  gc_ErrTranslation_fr_Texts : ARRAY[0..1193] OF POINTER TO WSTRING(101) := [ADR(gc_ErrTranslation_fr_Text0), ADR(gc_ErrTranslation_fr_Text1), ADR(gc_ErrTranslation_fr_Text2), ADR(gc_ErrTranslation_fr_Text3), ADR(gc_ErrTranslation_fr_Text4), ADR(gc_ErrTranslation_fr_Text5), ADR(gc_ErrTranslation_fr_Text6), ADR(gc_ErrTranslation_fr_Text7), ADR(gc_ErrTranslation_fr_Text8), ADR(gc_ErrTranslation_fr_Text9), ADR(gc_ErrTranslation_fr_Text10), ADR(gc_ErrTranslation_fr_Text11), ADR(gc_ErrTranslation_fr_Text12), ADR(gc_ErrTranslation_fr_Text13), ADR(gc_ErrTranslation_fr_Text14), ADR(gc_ErrTranslation_fr_Text15), ADR(gc_ErrTranslation_fr_Text16), ADR(gc_ErrTranslation_fr_Text17), ADR(gc_ErrTranslation_fr_Text18), ADR(gc_ErrTranslation_fr_Text19), ADR(gc_ErrTranslation_fr_Text20), ADR(gc_ErrTranslation_fr_Text21), ADR(gc_ErrTranslation_fr_Text22), ADR(gc_ErrTranslation_fr_Text23), ADR(gc_ErrTranslation_fr_Text24), ADR(gc_ErrTranslation_fr_Text25), ADR(gc_ErrTranslation_fr_Text26), ADR(gc_ErrTranslation_fr_Text27), ADR(gc_ErrTranslation_fr_Text28), ADR(gc_ErrTranslation_fr_Text29), ADR(gc_ErrTranslation_fr_Text30), ADR(gc_ErrTranslation_fr_Text31), ADR(gc_ErrTranslation_fr_Text32), ADR(gc_ErrTranslation_fr_Text33), ADR(gc_ErrTranslation_fr_Text34), ADR(gc_ErrTranslation_fr_Text35), ADR(gc_ErrTranslation_fr_Text36), ADR(gc_ErrTranslation_fr_Text37), ADR(gc_ErrTranslation_fr_Text38), ADR(gc_ErrTranslation_fr_Text39), ADR(gc_ErrTranslation_fr_Text40), ADR(gc_ErrTranslation_fr_Text41), ADR(gc_ErrTranslation_fr_Text42), ADR(gc_ErrTranslation_fr_Text43), ADR(gc_ErrTranslation_fr_Text44), ADR(gc_ErrTranslation_fr_Text45), ADR(gc_ErrTranslation_fr_Text46), ADR(gc_ErrTranslation_fr_Text47), ADR(gc_ErrTranslation_fr_Text48), ADR(gc_ErrTranslation_fr_Text49), ADR(gc_ErrTranslation_fr_Text50), ADR(gc_ErrTranslation_fr_Text51), ADR(gc_ErrTranslation_fr_Text52), ADR(gc_ErrTranslation_fr_Text53), ADR(gc_ErrTranslation_fr_Text54), ADR(gc_ErrTranslation_fr_Text55), ADR(gc_ErrTranslation_fr_Text56), ADR(gc_ErrTranslation_fr_Text57), ADR(gc_ErrTranslation_fr_Text58), ADR(gc_ErrTranslation_fr_Text59), ADR(gc_ErrTranslation_fr_Text60), ADR(gc_ErrTranslation_fr_Text61), ADR(gc_ErrTranslation_fr_Text62), ADR(gc_ErrTranslation_fr_Text63), ADR(gc_ErrTranslation_fr_Text64), ADR(gc_ErrTranslation_fr_Text65), ADR(gc_ErrTranslation_fr_Text66), ADR(gc_ErrTranslation_fr_Text67), ADR(gc_ErrTranslation_fr_Text68), ADR(gc_ErrTranslation_fr_Text69), ADR(gc_ErrTranslation_fr_Text70), ADR(gc_ErrTranslation_fr_Text71), ADR(gc_ErrTranslation_fr_Text72), ADR(gc_ErrTranslation_fr_Text73), ADR(gc_ErrTranslation_fr_Text74), ADR(gc_ErrTranslation_fr_Text75), ADR(gc_ErrTranslation_fr_Text76), ADR(gc_ErrTranslation_fr_Text77), ADR(gc_ErrTranslation_fr_Text78), ADR(gc_ErrTranslation_fr_Text79), ADR(gc_ErrTranslation_fr_Text80), ADR(gc_ErrTranslation_fr_Text81), ADR(gc_ErrTranslation_fr_Text82), ADR(gc_ErrTranslation_fr_Text83), ADR(gc_ErrTranslation_fr_Text84), ADR(gc_ErrTranslation_fr_Text85), ADR(gc_ErrTranslation_fr_Text86), ADR(gc_ErrTranslation_fr_Text87), ADR(gc_ErrTranslation_fr_Text88), ADR(gc_ErrTranslation_fr_Text89), ADR(gc_ErrTranslation_fr_Text90), ADR(gc_ErrTranslation_fr_Text91), ADR(gc_ErrTranslation_fr_Text92), ADR(gc_ErrTranslation_fr_Text93), ADR(gc_ErrTranslation_fr_Text94), ADR(gc_ErrTranslation_fr_Text95), ADR(gc_ErrTranslation_fr_Text96), ADR(gc_ErrTranslation_fr_Text97), ADR(gc_ErrTranslation_fr_Text98), ADR(gc_ErrTranslation_fr_Text99), ADR(gc_ErrTranslation_fr_Text100), ADR(gc_ErrTranslation_fr_Text101), ADR(gc_ErrTranslation_fr_Text102), ADR(gc_ErrTranslation_fr_Text103), ADR(gc_ErrTranslation_fr_Text104), ADR(gc_ErrTranslation_fr_Text105), ADR(gc_ErrTranslation_fr_Text106), ADR(gc_ErrTranslation_fr_Text107), ADR(gc_ErrTranslation_fr_Text108), ADR(gc_ErrTranslation_fr_Text109), ADR(gc_ErrTranslation_fr_Text110), ADR(gc_ErrTranslation_fr_Text111), ADR(gc_ErrTranslation_fr_Text112), ADR(gc_ErrTranslation_fr_Text113), ADR(gc_ErrTranslation_fr_Text114), ADR(gc_ErrTranslation_fr_Text115), ADR(gc_ErrTranslation_fr_Text116), ADR(gc_ErrTranslation_fr_Text117), ADR(gc_ErrTranslation_fr_Text118), ADR(gc_ErrTranslation_fr_Text119), ADR(gc_ErrTranslation_fr_Text120), ADR(gc_ErrTranslation_fr_Text121), ADR(gc_ErrTranslation_fr_Text122), ADR(gc_ErrTranslation_fr_Text123), ADR(gc_ErrTranslation_fr_Text124), ADR(gc_ErrTranslation_fr_Text125), ADR(gc_ErrTranslation_fr_Text126), ADR(gc_ErrTranslation_fr_Text127), ADR(gc_ErrTranslation_fr_Text128), ADR(gc_ErrTranslation_fr_Text129), ADR(gc_ErrTranslation_fr_Text130), ADR(gc_ErrTranslation_fr_Text131), ADR(gc_ErrTranslation_fr_Text132), ADR(gc_ErrTranslation_fr_Text133), ADR(gc_ErrTranslation_fr_Text134), ADR(gc_ErrTranslation_fr_Text135), ADR(gc_ErrTranslation_fr_Text136), ADR(gc_ErrTranslation_fr_Text137), ADR(gc_ErrTranslation_fr_Text138), ADR(gc_ErrTranslation_fr_Text139), ADR(gc_ErrTranslation_fr_Text140), ADR(gc_ErrTranslation_fr_Text141), ADR(gc_ErrTranslation_fr_Text142), ADR(gc_ErrTranslation_fr_Text143), ADR(gc_ErrTranslation_fr_Text144), ADR(gc_ErrTranslation_fr_Text145), ADR(gc_ErrTranslation_fr_Text146), ADR(gc_ErrTranslation_fr_Text147), ADR(gc_ErrTranslation_fr_Text148), ADR(gc_ErrTranslation_fr_Text149), ADR(gc_ErrTranslation_fr_Text150), ADR(gc_ErrTranslation_fr_Text151), ADR(gc_ErrTranslation_fr_Text152), ADR(gc_ErrTranslation_fr_Text153), ADR(gc_ErrTranslation_fr_Text154), ADR(gc_ErrTranslation_fr_Text155), ADR(gc_ErrTranslation_fr_Text156), ADR(gc_ErrTranslation_fr_Text157), ADR(gc_ErrTranslation_fr_Text158), ADR(gc_ErrTranslation_fr_Text159), ADR(gc_ErrTranslation_fr_Text160), ADR(gc_ErrTranslation_fr_Text161), ADR(gc_ErrTranslation_fr_Text162), ADR(gc_ErrTranslation_fr_Text163), ADR(gc_ErrTranslation_fr_Text164), ADR(gc_ErrTranslation_fr_Text165), ADR(gc_ErrTranslation_fr_Text166), ADR(gc_ErrTranslation_fr_Text167), ADR(gc_ErrTranslation_fr_Text168), ADR(gc_ErrTranslation_fr_Text169), ADR(gc_ErrTranslation_fr_Text170), ADR(gc_ErrTranslation_fr_Text171), ADR(gc_ErrTranslation_fr_Text172), ADR(gc_ErrTranslation_fr_Text173), ADR(gc_ErrTranslation_fr_Text174), ADR(gc_ErrTranslation_fr_Text175), ADR(gc_ErrTranslation_fr_Text176), ADR(gc_ErrTranslation_fr_Text177), ADR(gc_ErrTranslation_fr_Text178), ADR(gc_ErrTranslation_fr_Text179), ADR(gc_ErrTranslation_fr_Text180), ADR(gc_ErrTranslation_fr_Text181), ADR(gc_ErrTranslation_fr_Text182), ADR(gc_ErrTranslation_fr_Text183), ADR(gc_ErrTranslation_fr_Text184), ADR(gc_ErrTranslation_fr_Text185), ADR(gc_ErrTranslation_fr_Text186), ADR(gc_ErrTranslation_fr_Text187), ADR(gc_ErrTranslation_fr_Text188), ADR(gc_ErrTranslation_fr_Text189), ADR(gc_ErrTranslation_fr_Text190), ADR(gc_ErrTranslation_fr_Text191), ADR(gc_ErrTranslation_fr_Text192), ADR(gc_ErrTranslation_fr_Text193), ADR(gc_ErrTranslation_fr_Text194), ADR(gc_ErrTranslation_fr_Text195), ADR(gc_ErrTranslation_fr_Text196), ADR(gc_ErrTranslation_fr_Text197), ADR(gc_ErrTranslation_fr_Text198), ADR(gc_ErrTranslation_fr_Text199), ADR(gc_ErrTranslation_fr_Text200), ADR(gc_ErrTranslation_fr_Text201), ADR(gc_ErrTranslation_fr_Text202), ADR(gc_ErrTranslation_fr_Text203), ADR(gc_ErrTranslation_fr_Text204), ADR(gc_ErrTranslation_fr_Text205), ADR(gc_ErrTranslation_fr_Text206), ADR(gc_ErrTranslation_fr_Text207), ADR(gc_ErrTranslation_fr_Text208), ADR(gc_ErrTranslation_fr_Text209), ADR(gc_ErrTranslation_fr_Text210), ADR(gc_ErrTranslation_fr_Text211), ADR(gc_ErrTranslation_fr_Text212), ADR(gc_ErrTranslation_fr_Text213), ADR(gc_ErrTranslation_fr_Text214), ADR(gc_ErrTranslation_fr_Text215), ADR(gc_ErrTranslation_fr_Text216), ADR(gc_ErrTranslation_fr_Text217), ADR(gc_ErrTranslation_fr_Text218), ADR(gc_ErrTranslation_fr_Text219), ADR(gc_ErrTranslation_fr_Text220), ADR(gc_ErrTranslation_fr_Text221), ADR(gc_ErrTranslation_fr_Text222), ADR(gc_ErrTranslation_fr_Text223), ADR(gc_ErrTranslation_fr_Text224), ADR(gc_ErrTranslation_fr_Text225), ADR(gc_ErrTranslation_fr_Text226), ADR(gc_ErrTranslation_fr_Text227), ADR(gc_ErrTranslation_fr_Text228), ADR(gc_ErrTranslation_fr_Text229), ADR(gc_ErrTranslation_fr_Text230), ADR(gc_ErrTranslation_fr_Text231), ADR(gc_ErrTranslation_fr_Text232), ADR(gc_ErrTranslation_fr_Text233), ADR(gc_ErrTranslation_fr_Text234), ADR(gc_ErrTranslation_fr_Text235), ADR(gc_ErrTranslation_fr_Text236), ADR(gc_ErrTranslation_fr_Text237), ADR(gc_ErrTranslation_fr_Text238), ADR(gc_ErrTranslation_fr_Text239), ADR(gc_ErrTranslation_fr_Text240), ADR(gc_ErrTranslation_fr_Text241), ADR(gc_ErrTranslation_fr_Text242), ADR(gc_ErrTranslation_fr_Text243), ADR(gc_ErrTranslation_fr_Text244), ADR(gc_ErrTranslation_fr_Text245), ADR(gc_ErrTranslation_fr_Text246), ADR(gc_ErrTranslation_fr_Text247), ADR(gc_ErrTranslation_fr_Text248), ADR(gc_ErrTranslation_fr_Text249), ADR(gc_ErrTranslation_fr_Text250), ADR(gc_ErrTranslation_fr_Text251), ADR(gc_ErrTranslation_fr_Text252), ADR(gc_ErrTranslation_fr_Text253), ADR(gc_ErrTranslation_fr_Text254), ADR(gc_ErrTranslation_fr_Text255), ADR(gc_ErrTranslation_fr_Text256), ADR(gc_ErrTranslation_fr_Text257), ADR(gc_ErrTranslation_fr_Text258), ADR(gc_ErrTranslation_fr_Text259), ADR(gc_ErrTranslation_fr_Text260), ADR(gc_ErrTranslation_fr_Text261), ADR(gc_ErrTranslation_fr_Text262), ADR(gc_ErrTranslation_fr_Text263), ADR(gc_ErrTranslation_fr_Text264), ADR(gc_ErrTranslation_fr_Text265), ADR(gc_ErrTranslation_fr_Text266), ADR(gc_ErrTranslation_fr_Text267), ADR(gc_ErrTranslation_fr_Text268), ADR(gc_ErrTranslation_fr_Text269), ADR(gc_ErrTranslation_fr_Text270), ADR(gc_ErrTranslation_fr_Text271), ADR(gc_ErrTranslation_fr_Text272), ADR(gc_ErrTranslation_fr_Text273), ADR(gc_ErrTranslation_fr_Text274), ADR(gc_ErrTranslation_fr_Text275), ADR(gc_ErrTranslation_fr_Text276), ADR(gc_ErrTranslation_fr_Text277), ADR(gc_ErrTranslation_fr_Text278), ADR(gc_ErrTranslation_fr_Text279), ADR(gc_ErrTranslation_fr_Text280), ADR(gc_ErrTranslation_fr_Text281), ADR(gc_ErrTranslation_fr_Text282), ADR(gc_ErrTranslation_fr_Text283), ADR(gc_ErrTranslation_fr_Text284), ADR(gc_ErrTranslation_fr_Text285), ADR(gc_ErrTranslation_fr_Text286), ADR(gc_ErrTranslation_fr_Text287), ADR(gc_ErrTranslation_fr_Text288), ADR(gc_ErrTranslation_fr_Text289), ADR(gc_ErrTranslation_fr_Text290), ADR(gc_ErrTranslation_fr_Text291), ADR(gc_ErrTranslation_fr_Text292), ADR(gc_ErrTranslation_fr_Text293), ADR(gc_ErrTranslation_fr_Text294), ADR(gc_ErrTranslation_fr_Text295), ADR(gc_ErrTranslation_fr_Text296), ADR(gc_ErrTranslation_fr_Text297), ADR(gc_ErrTranslation_fr_Text298), ADR(gc_ErrTranslation_fr_Text299), ADR(gc_ErrTranslation_fr_Text300), ADR(gc_ErrTranslation_fr_Text301), ADR(gc_ErrTranslation_fr_Text302), ADR(gc_ErrTranslation_fr_Text303), ADR(gc_ErrTranslation_fr_Text304), ADR(gc_ErrTranslation_fr_Text305), ADR(gc_ErrTranslation_fr_Text306), ADR(gc_ErrTranslation_fr_Text307), ADR(gc_ErrTranslation_fr_Text308), ADR(gc_ErrTranslation_fr_Text309), ADR(gc_ErrTranslation_fr_Text310), ADR(gc_ErrTranslation_fr_Text311), ADR(gc_ErrTranslation_fr_Text312), ADR(gc_ErrTranslation_fr_Text313), ADR(gc_ErrTranslation_fr_Text314), ADR(gc_ErrTranslation_fr_Text315), ADR(gc_ErrTranslation_fr_Text316), ADR(gc_ErrTranslation_fr_Text317), ADR(gc_ErrTranslation_fr_Text318), ADR(gc_ErrTranslation_fr_Text319), ADR(gc_ErrTranslation_fr_Text320), ADR(gc_ErrTranslation_fr_Text321), ADR(gc_ErrTranslation_fr_Text322), ADR(gc_ErrTranslation_fr_Text323), ADR(gc_ErrTranslation_fr_Text324), ADR(gc_ErrTranslation_fr_Text325), ADR(gc_ErrTranslation_fr_Text326), ADR(gc_ErrTranslation_fr_Text327), ADR(gc_ErrTranslation_fr_Text328), ADR(gc_ErrTranslation_fr_Text329), ADR(gc_ErrTranslation_fr_Text330), ADR(gc_ErrTranslation_fr_Text331), ADR(gc_ErrTranslation_fr_Text332), ADR(gc_ErrTranslation_fr_Text333), ADR(gc_ErrTranslation_fr_Text334), ADR(gc_ErrTranslation_fr_Text335), ADR(gc_ErrTranslation_fr_Text336), ADR(gc_ErrTranslation_fr_Text337), ADR(gc_ErrTranslation_fr_Text338), ADR(gc_ErrTranslation_fr_Text339), ADR(gc_ErrTranslation_fr_Text340), ADR(gc_ErrTranslation_fr_Text341), ADR(gc_ErrTranslation_fr_Text342), ADR(gc_ErrTranslation_fr_Text343), ADR(gc_ErrTranslation_fr_Text344), ADR(gc_ErrTranslation_fr_Text345), ADR(gc_ErrTranslation_fr_Text346), ADR(gc_ErrTranslation_fr_Text347), ADR(gc_ErrTranslation_fr_Text348), ADR(gc_ErrTranslation_fr_Text349), ADR(gc_ErrTranslation_fr_Text350), ADR(gc_ErrTranslation_fr_Text351), ADR(gc_ErrTranslation_fr_Text352), ADR(gc_ErrTranslation_fr_Text353), ADR(gc_ErrTranslation_fr_Text354), ADR(gc_ErrTranslation_fr_Text355), ADR(gc_ErrTranslation_fr_Text356), ADR(gc_ErrTranslation_fr_Text357), ADR(gc_ErrTranslation_fr_Text358), ADR(gc_ErrTranslation_fr_Text359), ADR(gc_ErrTranslation_fr_Text360), ADR(gc_ErrTranslation_fr_Text361), ADR(gc_ErrTranslation_fr_Text362), ADR(gc_ErrTranslation_fr_Text363), ADR(gc_ErrTranslation_fr_Text364), ADR(gc_ErrTranslation_fr_Text365), ADR(gc_ErrTranslation_fr_Text366), ADR(gc_ErrTranslation_fr_Text367), ADR(gc_ErrTranslation_fr_Text368), ADR(gc_ErrTranslation_fr_Text369), ADR(gc_ErrTranslation_fr_Text370), ADR(gc_ErrTranslation_fr_Text371), ADR(gc_ErrTranslation_fr_Text372), ADR(gc_ErrTranslation_fr_Text373), ADR(gc_ErrTranslation_fr_Text374), ADR(gc_ErrTranslation_fr_Text375), ADR(gc_ErrTranslation_fr_Text376), ADR(gc_ErrTranslation_fr_Text377), ADR(gc_ErrTranslation_fr_Text378), ADR(gc_ErrTranslation_fr_Text379), ADR(gc_ErrTranslation_fr_Text380), ADR(gc_ErrTranslation_fr_Text381), ADR(gc_ErrTranslation_fr_Text382), ADR(gc_ErrTranslation_fr_Text383), ADR(gc_ErrTranslation_fr_Text384), ADR(gc_ErrTranslation_fr_Text385), ADR(gc_ErrTranslation_fr_Text386), ADR(gc_ErrTranslation_fr_Text387), ADR(gc_ErrTranslation_fr_Text388), ADR(gc_ErrTranslation_fr_Text389), ADR(gc_ErrTranslation_fr_Text390), ADR(gc_ErrTranslation_fr_Text391), ADR(gc_ErrTranslation_fr_Text392), ADR(gc_ErrTranslation_fr_Text393), ADR(gc_ErrTranslation_fr_Text394), ADR(gc_ErrTranslation_fr_Text395), ADR(gc_ErrTranslation_fr_Text396), ADR(gc_ErrTranslation_fr_Text397), ADR(gc_ErrTranslation_fr_Text398), ADR(gc_ErrTranslation_fr_Text399), ADR(gc_ErrTranslation_fr_Text400), ADR(gc_ErrTranslation_fr_Text401), ADR(gc_ErrTranslation_fr_Text402), ADR(gc_ErrTranslation_fr_Text403), ADR(gc_ErrTranslation_fr_Text404), ADR(gc_ErrTranslation_fr_Text405), ADR(gc_ErrTranslation_fr_Text406), ADR(gc_ErrTranslation_fr_Text407), ADR(gc_ErrTranslation_fr_Text408), ADR(gc_ErrTranslation_fr_Text409), ADR(gc_ErrTranslation_fr_Text410), ADR(gc_ErrTranslation_fr_Text411), ADR(gc_ErrTranslation_fr_Text412), ADR(gc_ErrTranslation_fr_Text413), ADR(gc_ErrTranslation_fr_Text414), ADR(gc_ErrTranslation_fr_Text415), ADR(gc_ErrTranslation_fr_Text416), ADR(gc_ErrTranslation_fr_Text417), ADR(gc_ErrTranslation_fr_Text418), ADR(gc_ErrTranslation_fr_Text419), ADR(gc_ErrTranslation_fr_Text420), ADR(gc_ErrTranslation_fr_Text421), ADR(gc_ErrTranslation_fr_Text422), ADR(gc_ErrTranslation_fr_Text423), ADR(gc_ErrTranslation_fr_Text424), ADR(gc_ErrTranslation_fr_Text425), ADR(gc_ErrTranslation_fr_Text426), ADR(gc_ErrTranslation_fr_Text427), ADR(gc_ErrTranslation_fr_Text428), ADR(gc_ErrTranslation_fr_Text429), ADR(gc_ErrTranslation_fr_Text430), ADR(gc_ErrTranslation_fr_Text431), ADR(gc_ErrTranslation_fr_Text432), ADR(gc_ErrTranslation_fr_Text433), ADR(gc_ErrTranslation_fr_Text434), ADR(gc_ErrTranslation_fr_Text435), ADR(gc_ErrTranslation_fr_Text436), ADR(gc_ErrTranslation_fr_Text437), ADR(gc_ErrTranslation_fr_Text438), ADR(gc_ErrTranslation_fr_Text439), ADR(gc_ErrTranslation_fr_Text440), ADR(gc_ErrTranslation_fr_Text441), ADR(gc_ErrTranslation_fr_Text442), ADR(gc_ErrTranslation_fr_Text443), ADR(gc_ErrTranslation_fr_Text444), ADR(gc_ErrTranslation_fr_Text445), ADR(gc_ErrTranslation_fr_Text446), ADR(gc_ErrTranslation_fr_Text447), ADR(gc_ErrTranslation_fr_Text448), ADR(gc_ErrTranslation_fr_Text449), ADR(gc_ErrTranslation_fr_Text450), ADR(gc_ErrTranslation_fr_Text451), ADR(gc_ErrTranslation_fr_Text452), ADR(gc_ErrTranslation_fr_Text453), ADR(gc_ErrTranslation_fr_Text454), ADR(gc_ErrTranslation_fr_Text455), ADR(gc_ErrTranslation_fr_Text456), ADR(gc_ErrTranslation_fr_Text457), ADR(gc_ErrTranslation_fr_Text458), ADR(gc_ErrTranslation_fr_Text459), ADR(gc_ErrTranslation_fr_Text460), ADR(gc_ErrTranslation_fr_Text461), ADR(gc_ErrTranslation_fr_Text462), ADR(gc_ErrTranslation_fr_Text463), ADR(gc_ErrTranslation_fr_Text464), ADR(gc_ErrTranslation_fr_Text465), ADR(gc_ErrTranslation_fr_Text466), ADR(gc_ErrTranslation_fr_Text467), ADR(gc_ErrTranslation_fr_Text468), ADR(gc_ErrTranslation_fr_Text469), ADR(gc_ErrTranslation_fr_Text470), ADR(gc_ErrTranslation_fr_Text471), ADR(gc_ErrTranslation_fr_Text472), ADR(gc_ErrTranslation_fr_Text473), ADR(gc_ErrTranslation_fr_Text474), ADR(gc_ErrTranslation_fr_Text475), ADR(gc_ErrTranslation_fr_Text476), ADR(gc_ErrTranslation_fr_Text477), ADR(gc_ErrTranslation_fr_Text478), ADR(gc_ErrTranslation_fr_Text479), ADR(gc_ErrTranslation_fr_Text480), ADR(gc_ErrTranslation_fr_Text481), ADR(gc_ErrTranslation_fr_Text482), ADR(gc_ErrTranslation_fr_Text483), ADR(gc_ErrTranslation_fr_Text484), ADR(gc_ErrTranslation_fr_Text485), ADR(gc_ErrTranslation_fr_Text486), ADR(gc_ErrTranslation_fr_Text487), ADR(gc_ErrTranslation_fr_Text488), ADR(gc_ErrTranslation_fr_Text489), ADR(gc_ErrTranslation_fr_Text490), ADR(gc_ErrTranslation_fr_Text491), ADR(gc_ErrTranslation_fr_Text492), ADR(gc_ErrTranslation_fr_Text493), ADR(gc_ErrTranslation_fr_Text494), ADR(gc_ErrTranslation_fr_Text495), ADR(gc_ErrTranslation_fr_Text496), ADR(gc_ErrTranslation_fr_Text497), ADR(gc_ErrTranslation_fr_Text498), ADR(gc_ErrTranslation_fr_Text499), ADR(gc_ErrTranslation_fr_Text500), ADR(gc_ErrTranslation_fr_Text501), ADR(gc_ErrTranslation_fr_Text502), ADR(gc_ErrTranslation_fr_Text503), ADR(gc_ErrTranslation_fr_Text504), ADR(gc_ErrTranslation_fr_Text505), ADR(gc_ErrTranslation_fr_Text506), ADR(gc_ErrTranslation_fr_Text507), ADR(gc_ErrTranslation_fr_Text508), ADR(gc_ErrTranslation_fr_Text509), ADR(gc_ErrTranslation_fr_Text510), ADR(gc_ErrTranslation_fr_Text511), ADR(gc_ErrTranslation_fr_Text512), ADR(gc_ErrTranslation_fr_Text513), ADR(gc_ErrTranslation_fr_Text514), ADR(gc_ErrTranslation_fr_Text515), ADR(gc_ErrTranslation_fr_Text516), ADR(gc_ErrTranslation_fr_Text517), ADR(gc_ErrTranslation_fr_Text518), ADR(gc_ErrTranslation_fr_Text519), ADR(gc_ErrTranslation_fr_Text520), ADR(gc_ErrTranslation_fr_Text521), ADR(gc_ErrTranslation_fr_Text522), ADR(gc_ErrTranslation_fr_Text523), ADR(gc_ErrTranslation_fr_Text524), ADR(gc_ErrTranslation_fr_Text525), ADR(gc_ErrTranslation_fr_Text526), ADR(gc_ErrTranslation_fr_Text527), ADR(gc_ErrTranslation_fr_Text528), ADR(gc_ErrTranslation_fr_Text529), ADR(gc_ErrTranslation_fr_Text530), ADR(gc_ErrTranslation_fr_Text531), ADR(gc_ErrTranslation_fr_Text532), ADR(gc_ErrTranslation_fr_Text533), ADR(gc_ErrTranslation_fr_Text534), ADR(gc_ErrTranslation_fr_Text535), ADR(gc_ErrTranslation_fr_Text536), ADR(gc_ErrTranslation_fr_Text537), ADR(gc_ErrTranslation_fr_Text538), ADR(gc_ErrTranslation_fr_Text539), ADR(gc_ErrTranslation_fr_Text540), ADR(gc_ErrTranslation_fr_Text541), ADR(gc_ErrTranslation_fr_Text542), ADR(gc_ErrTranslation_fr_Text543), ADR(gc_ErrTranslation_fr_Text544), ADR(gc_ErrTranslation_fr_Text545), ADR(gc_ErrTranslation_fr_Text546), ADR(gc_ErrTranslation_fr_Text547), ADR(gc_ErrTranslation_fr_Text548), ADR(gc_ErrTranslation_fr_Text549), ADR(gc_ErrTranslation_fr_Text550), ADR(gc_ErrTranslation_fr_Text551), ADR(gc_ErrTranslation_fr_Text552), ADR(gc_ErrTranslation_fr_Text553), ADR(gc_ErrTranslation_fr_Text554), ADR(gc_ErrTranslation_fr_Text555), ADR(gc_ErrTranslation_fr_Text556), ADR(gc_ErrTranslation_fr_Text557), ADR(gc_ErrTranslation_fr_Text558), ADR(gc_ErrTranslation_fr_Text559), ADR(gc_ErrTranslation_fr_Text560), ADR(gc_ErrTranslation_fr_Text561), ADR(gc_ErrTranslation_fr_Text562), ADR(gc_ErrTranslation_fr_Text563), ADR(gc_ErrTranslation_fr_Text564), ADR(gc_ErrTranslation_fr_Text565), ADR(gc_ErrTranslation_fr_Text566), ADR(gc_ErrTranslation_fr_Text567), ADR(gc_ErrTranslation_fr_Text568), ADR(gc_ErrTranslation_fr_Text569), ADR(gc_ErrTranslation_fr_Text570), ADR(gc_ErrTranslation_fr_Text571), ADR(gc_ErrTranslation_fr_Text572), ADR(gc_ErrTranslation_fr_Text573), ADR(gc_ErrTranslation_fr_Text574), ADR(gc_ErrTranslation_fr_Text575), ADR(gc_ErrTranslation_fr_Text576), ADR(gc_ErrTranslation_fr_Text577), ADR(gc_ErrTranslation_fr_Text578), ADR(gc_ErrTranslation_fr_Text579), ADR(gc_ErrTranslation_fr_Text580), ADR(gc_ErrTranslation_fr_Text581), ADR(gc_ErrTranslation_fr_Text582), ADR(gc_ErrTranslation_fr_Text583), ADR(gc_ErrTranslation_fr_Text584), ADR(gc_ErrTranslation_fr_Text585), ADR(gc_ErrTranslation_fr_Text586), ADR(gc_ErrTranslation_fr_Text587), ADR(gc_ErrTranslation_fr_Text588), ADR(gc_ErrTranslation_fr_Text589), ADR(gc_ErrTranslation_fr_Text590), ADR(gc_ErrTranslation_fr_Text591), ADR(gc_ErrTranslation_fr_Text592), ADR(gc_ErrTranslation_fr_Text593), ADR(gc_ErrTranslation_fr_Text594), ADR(gc_ErrTranslation_fr_Text595), ADR(gc_ErrTranslation_fr_Text596), ADR(gc_ErrTranslation_fr_Text597), ADR(gc_ErrTranslation_fr_Text598), ADR(gc_ErrTranslation_fr_Text599), ADR(gc_ErrTranslation_fr_Text600), ADR(gc_ErrTranslation_fr_Text601), ADR(gc_ErrTranslation_fr_Text602), ADR(gc_ErrTranslation_fr_Text603), ADR(gc_ErrTranslation_fr_Text604), ADR(gc_ErrTranslation_fr_Text605), ADR(gc_ErrTranslation_fr_Text606), ADR(gc_ErrTranslation_fr_Text607), ADR(gc_ErrTranslation_fr_Text608), ADR(gc_ErrTranslation_fr_Text609), ADR(gc_ErrTranslation_fr_Text610), ADR(gc_ErrTranslation_fr_Text611), ADR(gc_ErrTranslation_fr_Text612), ADR(gc_ErrTranslation_fr_Text613), ADR(gc_ErrTranslation_fr_Text614), ADR(gc_ErrTranslation_fr_Text615), ADR(gc_ErrTranslation_fr_Text616), ADR(gc_ErrTranslation_fr_Text617), ADR(gc_ErrTranslation_fr_Text618), ADR(gc_ErrTranslation_fr_Text619), ADR(gc_ErrTranslation_fr_Text620), ADR(gc_ErrTranslation_fr_Text621), ADR(gc_ErrTranslation_fr_Text622), ADR(gc_ErrTranslation_fr_Text623), ADR(gc_ErrTranslation_fr_Text624), ADR(gc_ErrTranslation_fr_Text625), ADR(gc_ErrTranslation_fr_Text626), ADR(gc_ErrTranslation_fr_Text627), ADR(gc_ErrTranslation_fr_Text628), ADR(gc_ErrTranslation_fr_Text629), ADR(gc_ErrTranslation_fr_Text630), ADR(gc_ErrTranslation_fr_Text631), ADR(gc_ErrTranslation_fr_Text632), ADR(gc_ErrTranslation_fr_Text633), ADR(gc_ErrTranslation_fr_Text634), ADR(gc_ErrTranslation_fr_Text635), ADR(gc_ErrTranslation_fr_Text636), ADR(gc_ErrTranslation_fr_Text637), ADR(gc_ErrTranslation_fr_Text638), ADR(gc_ErrTranslation_fr_Text639), ADR(gc_ErrTranslation_fr_Text640), ADR(gc_ErrTranslation_fr_Text641), ADR(gc_ErrTranslation_fr_Text642), ADR(gc_ErrTranslation_fr_Text643), ADR(gc_ErrTranslation_fr_Text644), ADR(gc_ErrTranslation_fr_Text645), ADR(gc_ErrTranslation_fr_Text646), ADR(gc_ErrTranslation_fr_Text647), ADR(gc_ErrTranslation_fr_Text648), ADR(gc_ErrTranslation_fr_Text649), ADR(gc_ErrTranslation_fr_Text650), ADR(gc_ErrTranslation_fr_Text651), ADR(gc_ErrTranslation_fr_Text652), ADR(gc_ErrTranslation_fr_Text653), ADR(gc_ErrTranslation_fr_Text654), ADR(gc_ErrTranslation_fr_Text655), ADR(gc_ErrTranslation_fr_Text656), ADR(gc_ErrTranslation_fr_Text657), ADR(gc_ErrTranslation_fr_Text658), ADR(gc_ErrTranslation_fr_Text659), ADR(gc_ErrTranslation_fr_Text660), ADR(gc_ErrTranslation_fr_Text661), ADR(gc_ErrTranslation_fr_Text662), ADR(gc_ErrTranslation_fr_Text663), ADR(gc_ErrTranslation_fr_Text664), ADR(gc_ErrTranslation_fr_Text665), ADR(gc_ErrTranslation_fr_Text666), ADR(gc_ErrTranslation_fr_Text667), ADR(gc_ErrTranslation_fr_Text668), ADR(gc_ErrTranslation_fr_Text669), ADR(gc_ErrTranslation_fr_Text670), ADR(gc_ErrTranslation_fr_Text671), ADR(gc_ErrTranslation_fr_Text672), ADR(gc_ErrTranslation_fr_Text673), ADR(gc_ErrTranslation_fr_Text674), ADR(gc_ErrTranslation_fr_Text675), ADR(gc_ErrTranslation_fr_Text676), ADR(gc_ErrTranslation_fr_Text677), ADR(gc_ErrTranslation_fr_Text678), ADR(gc_ErrTranslation_fr_Text679), ADR(gc_ErrTranslation_fr_Text680), ADR(gc_ErrTranslation_fr_Text681), ADR(gc_ErrTranslation_fr_Text682), ADR(gc_ErrTranslation_fr_Text683), ADR(gc_ErrTranslation_fr_Text684), ADR(gc_ErrTranslation_fr_Text685), ADR(gc_ErrTranslation_fr_Text686), ADR(gc_ErrTranslation_fr_Text687), ADR(gc_ErrTranslation_fr_Text688), ADR(gc_ErrTranslation_fr_Text689), ADR(gc_ErrTranslation_fr_Text690), ADR(gc_ErrTranslation_fr_Text691), ADR(gc_ErrTranslation_fr_Text692), ADR(gc_ErrTranslation_fr_Text693), ADR(gc_ErrTranslation_fr_Text694), ADR(gc_ErrTranslation_fr_Text695), ADR(gc_ErrTranslation_fr_Text696), ADR(gc_ErrTranslation_fr_Text697), ADR(gc_ErrTranslation_fr_Text698), ADR(gc_ErrTranslation_fr_Text699), ADR(gc_ErrTranslation_fr_Text700), ADR(gc_ErrTranslation_fr_Text701), ADR(gc_ErrTranslation_fr_Text702), ADR(gc_ErrTranslation_fr_Text703), ADR(gc_ErrTranslation_fr_Text704), ADR(gc_ErrTranslation_fr_Text705), ADR(gc_ErrTranslation_fr_Text706), ADR(gc_ErrTranslation_fr_Text707), ADR(gc_ErrTranslation_fr_Text708), ADR(gc_ErrTranslation_fr_Text709), ADR(gc_ErrTranslation_fr_Text710), ADR(gc_ErrTranslation_fr_Text711), ADR(gc_ErrTranslation_fr_Text712), ADR(gc_ErrTranslation_fr_Text713), ADR(gc_ErrTranslation_fr_Text714), ADR(gc_ErrTranslation_fr_Text715), ADR(gc_ErrTranslation_fr_Text716), ADR(gc_ErrTranslation_fr_Text717), ADR(gc_ErrTranslation_fr_Text718), ADR(gc_ErrTranslation_fr_Text719), ADR(gc_ErrTranslation_fr_Text720), ADR(gc_ErrTranslation_fr_Text721), ADR(gc_ErrTranslation_fr_Text722), ADR(gc_ErrTranslation_fr_Text723), ADR(gc_ErrTranslation_fr_Text724), ADR(gc_ErrTranslation_fr_Text725), ADR(gc_ErrTranslation_fr_Text726), ADR(gc_ErrTranslation_fr_Text727), ADR(gc_ErrTranslation_fr_Text728), ADR(gc_ErrTranslation_fr_Text729), ADR(gc_ErrTranslation_fr_Text730), ADR(gc_ErrTranslation_fr_Text731), ADR(gc_ErrTranslation_fr_Text732), ADR(gc_ErrTranslation_fr_Text733), ADR(gc_ErrTranslation_fr_Text734), ADR(gc_ErrTranslation_fr_Text735), ADR(gc_ErrTranslation_fr_Text736), ADR(gc_ErrTranslation_fr_Text737), ADR(gc_ErrTranslation_fr_Text738), ADR(gc_ErrTranslation_fr_Text739), ADR(gc_ErrTranslation_fr_Text740), ADR(gc_ErrTranslation_fr_Text741), ADR(gc_ErrTranslation_fr_Text742), ADR(gc_ErrTranslation_fr_Text743), ADR(gc_ErrTranslation_fr_Text744), ADR(gc_ErrTranslation_fr_Text745), ADR(gc_ErrTranslation_fr_Text746), ADR(gc_ErrTranslation_fr_Text747), ADR(gc_ErrTranslation_fr_Text748), ADR(gc_ErrTranslation_fr_Text749), ADR(gc_ErrTranslation_fr_Text750), ADR(gc_ErrTranslation_fr_Text751), ADR(gc_ErrTranslation_fr_Text752), ADR(gc_ErrTranslation_fr_Text753), ADR(gc_ErrTranslation_fr_Text754), ADR(gc_ErrTranslation_fr_Text755), ADR(gc_ErrTranslation_fr_Text756), ADR(gc_ErrTranslation_fr_Text757), ADR(gc_ErrTranslation_fr_Text758), ADR(gc_ErrTranslation_fr_Text759), ADR(gc_ErrTranslation_fr_Text760), ADR(gc_ErrTranslation_fr_Text761), ADR(gc_ErrTranslation_fr_Text762), ADR(gc_ErrTranslation_fr_Text763), ADR(gc_ErrTranslation_fr_Text764), ADR(gc_ErrTranslation_fr_Text765), ADR(gc_ErrTranslation_fr_Text766), ADR(gc_ErrTranslation_fr_Text767), ADR(gc_ErrTranslation_fr_Text768), ADR(gc_ErrTranslation_fr_Text769), ADR(gc_ErrTranslation_fr_Text770), ADR(gc_ErrTranslation_fr_Text771), ADR(gc_ErrTranslation_fr_Text772), ADR(gc_ErrTranslation_fr_Text773), ADR(gc_ErrTranslation_fr_Text774), ADR(gc_ErrTranslation_fr_Text775), ADR(gc_ErrTranslation_fr_Text776), ADR(gc_ErrTranslation_fr_Text777), ADR(gc_ErrTranslation_fr_Text778), ADR(gc_ErrTranslation_fr_Text779), ADR(gc_ErrTranslation_fr_Text780), ADR(gc_ErrTranslation_fr_Text781), ADR(gc_ErrTranslation_fr_Text782), ADR(gc_ErrTranslation_fr_Text783), ADR(gc_ErrTranslation_fr_Text784), ADR(gc_ErrTranslation_fr_Text785), ADR(gc_ErrTranslation_fr_Text786), ADR(gc_ErrTranslation_fr_Text787), ADR(gc_ErrTranslation_fr_Text788), ADR(gc_ErrTranslation_fr_Text789), ADR(gc_ErrTranslation_fr_Text790), ADR(gc_ErrTranslation_fr_Text791), ADR(gc_ErrTranslation_fr_Text792), ADR(gc_ErrTranslation_fr_Text793), ADR(gc_ErrTranslation_fr_Text794), ADR(gc_ErrTranslation_fr_Text795), ADR(gc_ErrTranslation_fr_Text796), ADR(gc_ErrTranslation_fr_Text797), ADR(gc_ErrTranslation_fr_Text798), ADR(gc_ErrTranslation_fr_Text799), ADR(gc_ErrTranslation_fr_Text800), ADR(gc_ErrTranslation_fr_Text801), ADR(gc_ErrTranslation_fr_Text802), ADR(gc_ErrTranslation_fr_Text803), ADR(gc_ErrTranslation_fr_Text804), ADR(gc_ErrTranslation_fr_Text805), ADR(gc_ErrTranslation_fr_Text806), ADR(gc_ErrTranslation_fr_Text807), ADR(gc_ErrTranslation_fr_Text808), ADR(gc_ErrTranslation_fr_Text809), ADR(gc_ErrTranslation_fr_Text810), ADR(gc_ErrTranslation_fr_Text811), ADR(gc_ErrTranslation_fr_Text812), ADR(gc_ErrTranslation_fr_Text813), ADR(gc_ErrTranslation_fr_Text814), ADR(gc_ErrTranslation_fr_Text815), ADR(gc_ErrTranslation_fr_Text816), ADR(gc_ErrTranslation_fr_Text817), ADR(gc_ErrTranslation_fr_Text818), ADR(gc_ErrTranslation_fr_Text819), ADR(gc_ErrTranslation_fr_Text820), ADR(gc_ErrTranslation_fr_Text821), ADR(gc_ErrTranslation_fr_Text822), ADR(gc_ErrTranslation_fr_Text823), ADR(gc_ErrTranslation_fr_Text824), ADR(gc_ErrTranslation_fr_Text825), ADR(gc_ErrTranslation_fr_Text826), ADR(gc_ErrTranslation_fr_Text827), ADR(gc_ErrTranslation_fr_Text828), ADR(gc_ErrTranslation_fr_Text829), ADR(gc_ErrTranslation_fr_Text830), ADR(gc_ErrTranslation_fr_Text831), ADR(gc_ErrTranslation_fr_Text832), ADR(gc_ErrTranslation_fr_Text833), ADR(gc_ErrTranslation_fr_Text834), ADR(gc_ErrTranslation_fr_Text835), ADR(gc_ErrTranslation_fr_Text836), ADR(gc_ErrTranslation_fr_Text837), ADR(gc_ErrTranslation_fr_Text838), ADR(gc_ErrTranslation_fr_Text839), ADR(gc_ErrTranslation_fr_Text840), ADR(gc_ErrTranslation_fr_Text841), ADR(gc_ErrTranslation_fr_Text842), ADR(gc_ErrTranslation_fr_Text843), ADR(gc_ErrTranslation_fr_Text844), ADR(gc_ErrTranslation_fr_Text845), ADR(gc_ErrTranslation_fr_Text846), ADR(gc_ErrTranslation_fr_Text847), ADR(gc_ErrTranslation_fr_Text848), ADR(gc_ErrTranslation_fr_Text849), ADR(gc_ErrTranslation_fr_Text850), ADR(gc_ErrTranslation_fr_Text851), ADR(gc_ErrTranslation_fr_Text852), ADR(gc_ErrTranslation_fr_Text853), ADR(gc_ErrTranslation_fr_Text854), ADR(gc_ErrTranslation_fr_Text855), ADR(gc_ErrTranslation_fr_Text856), ADR(gc_ErrTranslation_fr_Text857), ADR(gc_ErrTranslation_fr_Text858), ADR(gc_ErrTranslation_fr_Text859), ADR(gc_ErrTranslation_fr_Text860), ADR(gc_ErrTranslation_fr_Text861), ADR(gc_ErrTranslation_fr_Text862), ADR(gc_ErrTranslation_fr_Text863), ADR(gc_ErrTranslation_fr_Text864), ADR(gc_ErrTranslation_fr_Text865), ADR(gc_ErrTranslation_fr_Text866), ADR(gc_ErrTranslation_fr_Text867), ADR(gc_ErrTranslation_fr_Text868), ADR(gc_ErrTranslation_fr_Text869), ADR(gc_ErrTranslation_fr_Text870), ADR(gc_ErrTranslation_fr_Text871), ADR(gc_ErrTranslation_fr_Text872), ADR(gc_ErrTranslation_fr_Text873), ADR(gc_ErrTranslation_fr_Text874), ADR(gc_ErrTranslation_fr_Text875), ADR(gc_ErrTranslation_fr_Text876), ADR(gc_ErrTranslation_fr_Text877), ADR(gc_ErrTranslation_fr_Text878), ADR(gc_ErrTranslation_fr_Text879), ADR(gc_ErrTranslation_fr_Text880), ADR(gc_ErrTranslation_fr_Text881), ADR(gc_ErrTranslation_fr_Text882), ADR(gc_ErrTranslation_fr_Text883), ADR(gc_ErrTranslation_fr_Text884), ADR(gc_ErrTranslation_fr_Text885), ADR(gc_ErrTranslation_fr_Text886), ADR(gc_ErrTranslation_fr_Text887), ADR(gc_ErrTranslation_fr_Text888), ADR(gc_ErrTranslation_fr_Text889), ADR(gc_ErrTranslation_fr_Text890), ADR(gc_ErrTranslation_fr_Text891), ADR(gc_ErrTranslation_fr_Text892), ADR(gc_ErrTranslation_fr_Text893), ADR(gc_ErrTranslation_fr_Text894), ADR(gc_ErrTranslation_fr_Text895), ADR(gc_ErrTranslation_fr_Text896), ADR(gc_ErrTranslation_fr_Text897), ADR(gc_ErrTranslation_fr_Text898), ADR(gc_ErrTranslation_fr_Text899), ADR(gc_ErrTranslation_fr_Text900), ADR(gc_ErrTranslation_fr_Text901), ADR(gc_ErrTranslation_fr_Text902), ADR(gc_ErrTranslation_fr_Text903), ADR(gc_ErrTranslation_fr_Text904), ADR(gc_ErrTranslation_fr_Text905), ADR(gc_ErrTranslation_fr_Text906), ADR(gc_ErrTranslation_fr_Text907), ADR(gc_ErrTranslation_fr_Text908), ADR(gc_ErrTranslation_fr_Text909), ADR(gc_ErrTranslation_fr_Text910), ADR(gc_ErrTranslation_fr_Text911), ADR(gc_ErrTranslation_fr_Text912), ADR(gc_ErrTranslation_fr_Text913), ADR(gc_ErrTranslation_fr_Text914), ADR(gc_ErrTranslation_fr_Text915), ADR(gc_ErrTranslation_fr_Text916), ADR(gc_ErrTranslation_fr_Text917), ADR(gc_ErrTranslation_fr_Text918), ADR(gc_ErrTranslation_fr_Text919), ADR(gc_ErrTranslation_fr_Text920), ADR(gc_ErrTranslation_fr_Text921), ADR(gc_ErrTranslation_fr_Text922), ADR(gc_ErrTranslation_fr_Text923), ADR(gc_ErrTranslation_fr_Text924), ADR(gc_ErrTranslation_fr_Text925), ADR(gc_ErrTranslation_fr_Text926), ADR(gc_ErrTranslation_fr_Text927), ADR(gc_ErrTranslation_fr_Text928), ADR(gc_ErrTranslation_fr_Text929), ADR(gc_ErrTranslation_fr_Text930), ADR(gc_ErrTranslation_fr_Text931), ADR(gc_ErrTranslation_fr_Text932), ADR(gc_ErrTranslation_fr_Text933), ADR(gc_ErrTranslation_fr_Text934), ADR(gc_ErrTranslation_fr_Text935), ADR(gc_ErrTranslation_fr_Text936), ADR(gc_ErrTranslation_fr_Text937), ADR(gc_ErrTranslation_fr_Text938), ADR(gc_ErrTranslation_fr_Text939), ADR(gc_ErrTranslation_fr_Text940), ADR(gc_ErrTranslation_fr_Text941), ADR(gc_ErrTranslation_fr_Text942), ADR(gc_ErrTranslation_fr_Text943), ADR(gc_ErrTranslation_fr_Text944), ADR(gc_ErrTranslation_fr_Text945), ADR(gc_ErrTranslation_fr_Text946), ADR(gc_ErrTranslation_fr_Text947), ADR(gc_ErrTranslation_fr_Text948), ADR(gc_ErrTranslation_fr_Text949), ADR(gc_ErrTranslation_fr_Text950), ADR(gc_ErrTranslation_fr_Text951), ADR(gc_ErrTranslation_fr_Text952), ADR(gc_ErrTranslation_fr_Text953), ADR(gc_ErrTranslation_fr_Text954), ADR(gc_ErrTranslation_fr_Text955), ADR(gc_ErrTranslation_fr_Text956), ADR(gc_ErrTranslation_fr_Text957), ADR(gc_ErrTranslation_fr_Text958), ADR(gc_ErrTranslation_fr_Text959), ADR(gc_ErrTranslation_fr_Text960), ADR(gc_ErrTranslation_fr_Text961), ADR(gc_ErrTranslation_fr_Text962), ADR(gc_ErrTranslation_fr_Text963), ADR(gc_ErrTranslation_fr_Text964), ADR(gc_ErrTranslation_fr_Text965), ADR(gc_ErrTranslation_fr_Text966), ADR(gc_ErrTranslation_fr_Text967), ADR(gc_ErrTranslation_fr_Text968), ADR(gc_ErrTranslation_fr_Text969), ADR(gc_ErrTranslation_fr_Text970), ADR(gc_ErrTranslation_fr_Text971), ADR(gc_ErrTranslation_fr_Text972), ADR(gc_ErrTranslation_fr_Text973), ADR(gc_ErrTranslation_fr_Text974), ADR(gc_ErrTranslation_fr_Text975), ADR(gc_ErrTranslation_fr_Text976), ADR(gc_ErrTranslation_fr_Text977), ADR(gc_ErrTranslation_fr_Text978), ADR(gc_ErrTranslation_fr_Text979), ADR(gc_ErrTranslation_fr_Text980), ADR(gc_ErrTranslation_fr_Text981), ADR(gc_ErrTranslation_fr_Text982), ADR(gc_ErrTranslation_fr_Text983), ADR(gc_ErrTranslation_fr_Text984), ADR(gc_ErrTranslation_fr_Text985), ADR(gc_ErrTranslation_fr_Text986), ADR(gc_ErrTranslation_fr_Text987), ADR(gc_ErrTranslation_fr_Text988), ADR(gc_ErrTranslation_fr_Text989), ADR(gc_ErrTranslation_fr_Text990), ADR(gc_ErrTranslation_fr_Text991), ADR(gc_ErrTranslation_fr_Text992), ADR(gc_ErrTranslation_fr_Text993), ADR(gc_ErrTranslation_fr_Text994), ADR(gc_ErrTranslation_fr_Text995), ADR(gc_ErrTranslation_fr_Text996), ADR(gc_ErrTranslation_fr_Text997), ADR(gc_ErrTranslation_fr_Text998), ADR(gc_ErrTranslation_fr_Text999), ADR(gc_ErrTranslation_fr_Text1000), ADR(gc_ErrTranslation_fr_Text1001), ADR(gc_ErrTranslation_fr_Text1002), ADR(gc_ErrTranslation_fr_Text1003), ADR(gc_ErrTranslation_fr_Text1004), ADR(gc_ErrTranslation_fr_Text1005), ADR(gc_ErrTranslation_fr_Text1006), ADR(gc_ErrTranslation_fr_Text1007), ADR(gc_ErrTranslation_fr_Text1008), ADR(gc_ErrTranslation_fr_Text1009), ADR(gc_ErrTranslation_fr_Text1010), ADR(gc_ErrTranslation_fr_Text1011), ADR(gc_ErrTranslation_fr_Text1012), ADR(gc_ErrTranslation_fr_Text1013), ADR(gc_ErrTranslation_fr_Text1014), ADR(gc_ErrTranslation_fr_Text1015), ADR(gc_ErrTranslation_fr_Text1016), ADR(gc_ErrTranslation_fr_Text1017), ADR(gc_ErrTranslation_fr_Text1018), ADR(gc_ErrTranslation_fr_Text1019), ADR(gc_ErrTranslation_fr_Text1020), ADR(gc_ErrTranslation_fr_Text1021), ADR(gc_ErrTranslation_fr_Text1022), ADR(gc_ErrTranslation_fr_Text1023), ADR(gc_ErrTranslation_fr_Text1024), ADR(gc_ErrTranslation_fr_Text1025), ADR(gc_ErrTranslation_fr_Text1026), ADR(gc_ErrTranslation_fr_Text1027), ADR(gc_ErrTranslation_fr_Text1028), ADR(gc_ErrTranslation_fr_Text1029), ADR(gc_ErrTranslation_fr_Text1030), ADR(gc_ErrTranslation_fr_Text1031), ADR(gc_ErrTranslation_fr_Text1032), ADR(gc_ErrTranslation_fr_Text1033), ADR(gc_ErrTranslation_fr_Text1034), ADR(gc_ErrTranslation_fr_Text1035), ADR(gc_ErrTranslation_fr_Text1036), ADR(gc_ErrTranslation_fr_Text1037), ADR(gc_ErrTranslation_fr_Text1038), ADR(gc_ErrTranslation_fr_Text1039), ADR(gc_ErrTranslation_fr_Text1040), ADR(gc_ErrTranslation_fr_Text1041), ADR(gc_ErrTranslation_fr_Text1042), ADR(gc_ErrTranslation_fr_Text1043), ADR(gc_ErrTranslation_fr_Text1044), ADR(gc_ErrTranslation_fr_Text1045), ADR(gc_ErrTranslation_fr_Text1046), ADR(gc_ErrTranslation_fr_Text1047), ADR(gc_ErrTranslation_fr_Text1048), ADR(gc_ErrTranslation_fr_Text1049), ADR(gc_ErrTranslation_fr_Text1050), ADR(gc_ErrTranslation_fr_Text1051), ADR(gc_ErrTranslation_fr_Text1052), ADR(gc_ErrTranslation_fr_Text1053), ADR(gc_ErrTranslation_fr_Text1054), ADR(gc_ErrTranslation_fr_Text1055), ADR(gc_ErrTranslation_fr_Text1056), ADR(gc_ErrTranslation_fr_Text1057), ADR(gc_ErrTranslation_fr_Text1058), ADR(gc_ErrTranslation_fr_Text1059), ADR(gc_ErrTranslation_fr_Text1060), ADR(gc_ErrTranslation_fr_Text1061), ADR(gc_ErrTranslation_fr_Text1062), ADR(gc_ErrTranslation_fr_Text1063), ADR(gc_ErrTranslation_fr_Text1064), ADR(gc_ErrTranslation_fr_Text1065), ADR(gc_ErrTranslation_fr_Text1066), ADR(gc_ErrTranslation_fr_Text1067), ADR(gc_ErrTranslation_fr_Text1068), ADR(gc_ErrTranslation_fr_Text1069), ADR(gc_ErrTranslation_fr_Text1070), ADR(gc_ErrTranslation_fr_Text1071), ADR(gc_ErrTranslation_fr_Text1072), ADR(gc_ErrTranslation_fr_Text1073), ADR(gc_ErrTranslation_fr_Text1074), ADR(gc_ErrTranslation_fr_Text1075), ADR(gc_ErrTranslation_fr_Text1076), ADR(gc_ErrTranslation_fr_Text1077), ADR(gc_ErrTranslation_fr_Text1078), ADR(gc_ErrTranslation_fr_Text1079), ADR(gc_ErrTranslation_fr_Text1080), ADR(gc_ErrTranslation_fr_Text1081), ADR(gc_ErrTranslation_fr_Text1082), ADR(gc_ErrTranslation_fr_Text1083), ADR(gc_ErrTranslation_fr_Text1084), ADR(gc_ErrTranslation_fr_Text1085), ADR(gc_ErrTranslation_fr_Text1086), ADR(gc_ErrTranslation_fr_Text1087), ADR(gc_ErrTranslation_fr_Text1088), ADR(gc_ErrTranslation_fr_Text1089), ADR(gc_ErrTranslation_fr_Text1090), ADR(gc_ErrTranslation_fr_Text1091), ADR(gc_ErrTranslation_fr_Text1092), ADR(gc_ErrTranslation_fr_Text1093), ADR(gc_ErrTranslation_fr_Text1094), ADR(gc_ErrTranslation_fr_Text1095), ADR(gc_ErrTranslation_fr_Text1096), ADR(gc_ErrTranslation_fr_Text1097), ADR(gc_ErrTranslation_fr_Text1098), ADR(gc_ErrTranslation_fr_Text1099), ADR(gc_ErrTranslation_fr_Text1100), ADR(gc_ErrTranslation_fr_Text1101), ADR(gc_ErrTranslation_fr_Text1102), ADR(gc_ErrTranslation_fr_Text1103), ADR(gc_ErrTranslation_fr_Text1104), ADR(gc_ErrTranslation_fr_Text1105), ADR(gc_ErrTranslation_fr_Text1106), ADR(gc_ErrTranslation_fr_Text1107), ADR(gc_ErrTranslation_fr_Text1108), ADR(gc_ErrTranslation_fr_Text1109), ADR(gc_ErrTranslation_fr_Text1110), ADR(gc_ErrTranslation_fr_Text1111), ADR(gc_ErrTranslation_fr_Text1112), ADR(gc_ErrTranslation_fr_Text1113), ADR(gc_ErrTranslation_fr_Text1114), ADR(gc_ErrTranslation_fr_Text1115), ADR(gc_ErrTranslation_fr_Text1116), ADR(gc_ErrTranslation_fr_Text1117), ADR(gc_ErrTranslation_fr_Text1118), ADR(gc_ErrTranslation_fr_Text1119), ADR(gc_ErrTranslation_fr_Text1120), ADR(gc_ErrTranslation_fr_Text1121), ADR(gc_ErrTranslation_fr_Text1122), ADR(gc_ErrTranslation_fr_Text1123), ADR(gc_ErrTranslation_fr_Text1124), ADR(gc_ErrTranslation_fr_Text1125), ADR(gc_ErrTranslation_fr_Text1126), ADR(gc_ErrTranslation_fr_Text1127), ADR(gc_ErrTranslation_fr_Text1128), ADR(gc_ErrTranslation_fr_Text1129), ADR(gc_ErrTranslation_fr_Text1130), ADR(gc_ErrTranslation_fr_Text1131), ADR(gc_ErrTranslation_fr_Text1132), ADR(gc_ErrTranslation_fr_Text1133), ADR(gc_ErrTranslation_fr_Text1134), ADR(gc_ErrTranslation_fr_Text1135), ADR(gc_ErrTranslation_fr_Text1136), ADR(gc_ErrTranslation_fr_Text1137), ADR(gc_ErrTranslation_fr_Text1138), ADR(gc_ErrTranslation_fr_Text1139), ADR(gc_ErrTranslation_fr_Text1140), ADR(gc_ErrTranslation_fr_Text1141), ADR(gc_ErrTranslation_fr_Text1142), ADR(gc_ErrTranslation_fr_Text1143), ADR(gc_ErrTranslation_fr_Text1144), ADR(gc_ErrTranslation_fr_Text1145), ADR(gc_ErrTranslation_fr_Text1146), ADR(gc_ErrTranslation_fr_Text1147), ADR(gc_ErrTranslation_fr_Text1148), ADR(gc_ErrTranslation_fr_Text1149), ADR(gc_ErrTranslation_fr_Text1150), ADR(gc_ErrTranslation_fr_Text1151), ADR(gc_ErrTranslation_fr_Text1152), ADR(gc_ErrTranslation_fr_Text1153), ADR(gc_ErrTranslation_fr_Text1154), ADR(gc_ErrTranslation_fr_Text1155), ADR(gc_ErrTranslation_fr_Text1156), ADR(gc_ErrTranslation_fr_Text1157), ADR(gc_ErrTranslation_fr_Text1158), ADR(gc_ErrTranslation_fr_Text1159), ADR(gc_ErrTranslation_fr_Text1160), ADR(gc_ErrTranslation_fr_Text1161), ADR(gc_ErrTranslation_fr_Text1162), ADR(gc_ErrTranslation_fr_Text1163), ADR(gc_ErrTranslation_fr_Text1164), ADR(gc_ErrTranslation_fr_Text1165), ADR(gc_ErrTranslation_fr_Text1166), ADR(gc_ErrTranslation_fr_Text1167), ADR(gc_ErrTranslation_fr_Text1168), ADR(gc_ErrTranslation_fr_Text1169), ADR(gc_ErrTranslation_fr_Text1170), ADR(gc_ErrTranslation_fr_Text1171), ADR(gc_ErrTranslation_fr_Text1172), ADR(gc_ErrTranslation_fr_Text1173), ADR(gc_ErrTranslation_fr_Text1174), ADR(gc_ErrTranslation_fr_Text1175), ADR(gc_ErrTranslation_fr_Text1176), ADR(gc_ErrTranslation_fr_Text1177), ADR(gc_ErrTranslation_fr_Text1178), ADR(gc_ErrTranslation_fr_Text1179), ADR(gc_ErrTranslation_fr_Text1180), ADR(gc_ErrTranslation_fr_Text1181), ADR(gc_ErrTranslation_fr_Text1182), ADR(gc_ErrTranslation_fr_Text1183), ADR(gc_ErrTranslation_fr_Text1184), ADR(gc_ErrTranslation_fr_Text1185), ADR(gc_ErrTranslation_fr_Text1186), ADR(gc_ErrTranslation_fr_Text1187), ADR(gc_ErrTranslation_fr_Text1188), ADR(gc_ErrTranslation_fr_Text1189), ADR(gc_ErrTranslation_fr_Text1190), ADR(gc_ErrTranslation_fr_Text1191), ADR(gc_ErrTranslation_fr_Text1192), ADR(gc_ErrTranslation_fr_Text1193)];
  gc_ErrTranslation_fr : TTranslation := (IsoCode := 'fr', EnglishName := "french", NativeName := "french", Texts := ADR(gc_ErrTranslation_fr_Texts));
  ERR_TRANSLATION_TEXT_COUNT : UINT := 1194;
  g_ErrTranslations : ARRAY[0..2] OF POINTER TO TTranslation := [ADR(gc_ErrTranslation_de), ADR(gc_ErrTranslation_en), ADR(gc_ErrTranslation_fr)];
END_VAR
